(* IEC 61131-3 sources: our-getting-started/test, 4 files *)

(* ---- testAdd.st ---- *)
USING AxUnit.Assert;
USING Siemens.Ax;

NAMESPACE Test
    {TestFixture}
    CLASS TestInt
        // Parametrized tests
        {Test(v1 := 1, v2 := 2, expectedResult := 3)}
        {Test(v1 := -1, v2 := 1, expectedResult := 0)}
        {Test(v1 := 32000, v2 := 32000, expectedResult := DINT#64000)}
        METHOD PUBLIC TestAddWithInts
            VAR_INPUT
                v1 : INT;
                v2 : INT;
                expectedResult : DINT;
            END_VAR
            Equal(expected := expectedResult, actual := Add(v1, v2));

        END_METHOD
    END_CLASS
END_NAMESPACE

(* ---- testHelloWorld.st ---- *)
USING AxUnit;
USING Siemens.Ax;

NAMESPACE Test

    {TestFixture}
    CLASS testHelloWorld
        {Test}
        METHOD PUBLIC MyTestMethod
            VAR_EXTERNAL
                myString : String;
            END_VAR
            Assert.Equal(actual := HelloWorldFunction(), expected := 'Hello AX World');
        END_METHOD
    END_CLASS

END_NAMESPACE

(* ---- testOperatingModeController.st ---- *)
USING AxUnit.Assert;
USING AxUnit;
USING Siemens.Ax;

NAMESPACE Test

    {TestFixture}
    CLASS testOperatingModeController
        VAR
            o : OperatingModeController := (Zone := 1);
        END_VAR
        {Test}
        METHOD PUBLIC GetOperatingMode_returns_Automatic
            o.SetOperatingMode(OperatingMode#Automatic);
            Equal(expected := TRUE, actual := o.GetOperatingMode() = OperatingMode#Automatic);
        END_METHOD
    END_CLASS

END_NAMESPACE

(* ---- testOperatingModeControllerExt.st ---- *)
USING AxUnit.Assert;
USING AxUnit;
USING Siemens.Ax;

NAMESPACE Test
    {TestFixture}
    CLASS testOperatingModeControllerExt
        VAR
            o : OperatingModeControllerExt := (Zone := 1);
        END_VAR
        {Test}
        METHOD PUBLIC GetZoneValueReturns_0_in_Maintenance_Mode;
            o.SetOperatingMode(OperatingMode#Manual);
            Equal(expected := FALSE, actual := o.GetZoneStatusAsInt() = 0);
            o.SetOperatingMode(OperatingMode#Maintenance);
            Equal(expected := 0, actual := o.GetZoneStatusAsInt());
        END_METHOD
    END_CLASS
END_NAMESPACE
